FUNCTION_BLOCK ParametersSelector (* Basic Function Block Type *)
  (* Standard: 61499-2 *)
  (* Version 0.0, 7/3/2024, SESA713705, Schneider Electric, Template *)
  PACKAGE SE.Nereda;
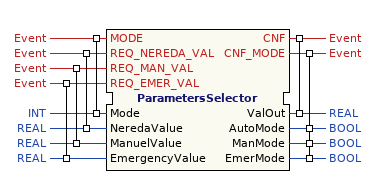
  EVENT_INPUT
    MODE WITH Mode;
    REQ_NEREDA_VAL WITH NeredaValue;
    REQ_MAN_VAL WITH ManuelValue;
    REQ_EMER_VAL WITH EmergencyValue;
  END_EVENT
  EVENT_OUTPUT
    CNF WITH ValOut; (* Execution Confirmation *)
    CNF_MODE WITH ManMode, AutoMode, EmerMode;
  END_EVENT
  VAR_INPUT
    Mode : INT;
    NeredaValue : REAL;
    ManuelValue : REAL;
    EmergencyValue : REAL;
  END_VAR
  VAR_OUTPUT
    ValOut : REAL;
    AutoMode : BOOL;
    ManMode : BOOL;
    EmerMode : BOOL;
  END_VAR
  VAR
    InValue : REAL;
  END_VAR
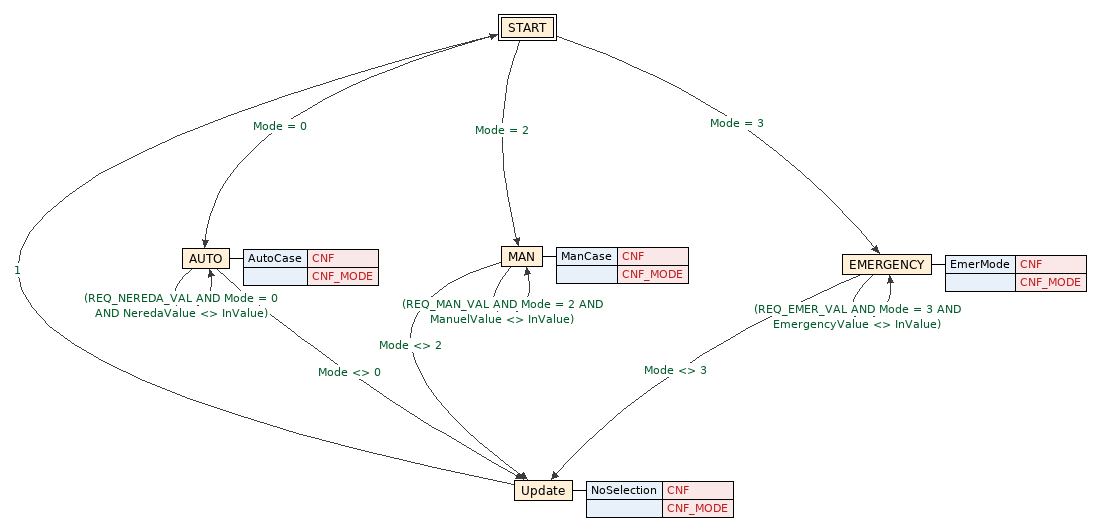
  EC_STATES
    START; (* Initial State *)
    AUTO : AutoCase -> CNF, -> CNF_MODE;
    MAN : ManCase -> CNF, -> CNF_MODE;
    EMERGENCY : EmerMode -> CNF, -> CNF_MODE;
    Update : NoSelection -> CNF, -> CNF_MODE;
  END_STATES
  EC_TRANSITIONS
    START TO AUTO := Mode = 0;
    START TO MAN := Mode = 2;
    AUTO TO AUTO := (REQ_NEREDA_VAL AND Mode = 0 AND NeredaValue <> InValue);
    MAN TO MAN := (REQ_MAN_VAL AND Mode = 2 AND ManuelValue <> InValue);
    START TO EMERGENCY := Mode = 3;
    EMERGENCY TO EMERGENCY := (REQ_EMER_VAL AND Mode = 3 AND EmergencyValue <> InValue);
    Update TO START := 1;
    MAN TO Update := Mode <> 2;
    AUTO TO Update := Mode <> 0;
    EMERGENCY TO Update := Mode <> 3;
  END_TRANSITIONS
  ALGORITHM AutoCase IN ST:
;
ValOut := NeredaValue;
InValue := NeredaValue;
AutoMode := TRUE;
ManMode := FALSE;
EmerMode := FALSE;
  END_ALGORITHM
  ALGORITHM ManCase IN ST:
;

ValOut := ManuelValue;
InValue := ManuelValue;
AutoMode := FALSE;
ManMode := TRUE;
EmerMode := FALSE;
  END_ALGORITHM
  ALGORITHM EmerMode IN ST:
;
ValOut := EmergencyValue;
InValue := EmergencyValue;
AutoMode := FALSE;
ManMode := FALSE;
EmerMode := TRUE;
  END_ALGORITHM
  ALGORITHM NoSelection IN ST:
;
ValOut := 0;
InValue := 0;
AutoMode := FALSE;
ManMode := FALSE;
EmerMode := FALSE;
  END_ALGORITHM
END_FUNCTION_BLOCK
